TYPE E_ReadBeamDataState :
(
	INIT,
	REQUEST_DATA,
	DATA_READY,
	MEASUREMENT_DONE,
	ERROR
);
END_TYPE

(* stored: Version 1.1.0.1, ProductVersion 3.1.4020.6
   DUT E_ReadBeamDataState: Id {c483b717-391e-4601-9066-9dd5283aaf7a} *)
